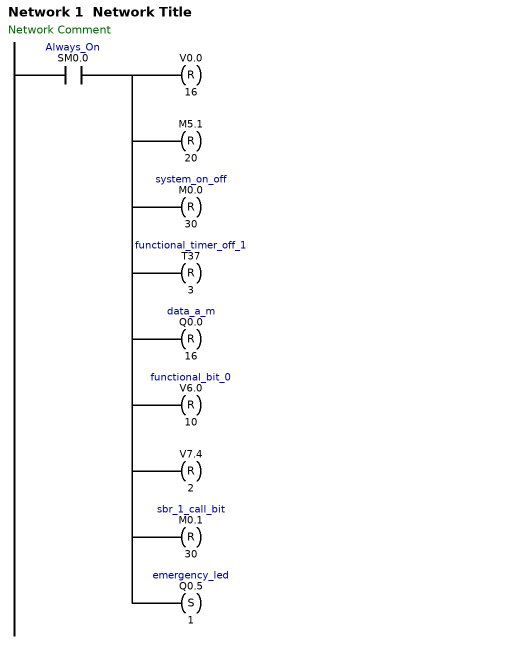
[picture p24: SBR15 networks 1-1]
Network 1 // Network Title
// Network Comment
LD     Always_On:SM0.0
R      V0.0, 16
R      M5.1, 20
R      system_on_off:M0.0, 30
R      functional_timer_off_1:T37, 3
R      data_a_m:Q0.0, 16
R      functional_bit_0:V6.0, 10
R      V7.4, 2
R      sbr_1_call_bit:M0.1, 30
S      emergency_led:Q0.5, 1
END_SUBROUTINE_BLOCK
